// TIA Portal V17 export
// export: Created 2023-02-13T11:16:22.7562679Z, ExportSetting WithDefaults, DisplayName Totally Integrated Automation Portal, DisplayVersion V17, DisplayName TIA Portal Openness, DisplayVersion V17, DisplayName TIA Portal Teamcenter Gateway, DisplayVersion V17, DisplayName TIA Portal Version Control Interface, DisplayVersion V17, DisplayName SINAMICS Startdrive Advanced, DisplayVersion V17, DisplayName SINAMICS Startdrive G130, G150, S120, S150, SINAMICS MV, S210, DisplayVersion V17, DisplayName SINAMICS Startdrive G110M, G120, G120C, G120D, G120P, G115D, DisplayVersion V17, DisplayName STEP 7 Professional, DisplayVersion V17, DisplayName STEP 7 Safety, DisplayVersion V17, DisplayName WinCC Professional, DisplayVersion V17
DATA_BLOCK "IO_Valve_Blend41_DB"   // DB62
VERSION : 0.1
// stored: AutoNumber true, DBAccessibleFromOPCUA true, DBAccessibleFromWebserver true, InstanceOfName IO_Valve_Blend41, InstanceOfType FB
"IO_Valve_Blend41"
   // VAR_INPUT
   //    "lock 1" : Bool;
   //    "lock 2" : Bool;
   //    "lock 3" : Bool;
   //    "lock 4" : Bool;
   //    init : Bool;
   //    reset : Bool;
   //    testing : Bool;
   // END_VAR
   // VAR
   //    "AV-41.01" : "Valve";
   //    "AV-41.02" : "Valve";
   //    "AV-41.03" : "Valve";
   //    "AV-41.04" : "Valve";
   //    "AV-41.05" : "Valve";
   //    "AV-41.06" : "Valve";
   //    "AV-41.07" : "Valve";
   //    "AV-41.08" : "Valve";
   //    "AV-41.09" : "Valve";
   //    "AV-41.10" : "Valve";
   //    "AV-41.11" : "Valve";
   //    "AV-41.12" : "Valve";
   //    "AV-41.13" : "Valve";
   //    "AV-41.14" : "Valve";
   //    "AV-41.15" : "Valve";
   //    "AV-41.16" : "Valve";
   //    "AV-41.17" : "Valve";
   //    "AV-41.18" : "Valve";
   //    "AV-41.19" : "Valve";
   //    "AV-41.20" : "Valve";
   //    "AV-41.21" : "Valve";
   //    "AV-41.22" : "Valve";
   //    "AV-41.23" : "Valve";
   //    "AV-41.24" : "Valve";
   //    "AV-41.25" : "Valve";
   //    "AV-41.26" : "Valve";
   //    "AV-41.27" : "Valve";
   //    "AV-41.28" : "Valve";
   //    "AV-41.29" : "Valve";
   //    "AV-41.30" : "Valve";
   //    "AV-41.31" : "Valve";
   //    "AV-41.32" : "Valve";
   //    "AV-41.33" : "Valve";
   //    "AV-41.34" : "Valve";
   // END_VAR
BEGIN
END_DATA_BLOCK
